{attribute 'linkalways'} 
{attribute 'no_explicit_call' := 'This FB is a CLASS and must be accessed using methods or properties'}
{attribute 'enable_dynamic_creation'}
FUNCTION_BLOCK _ETcVnEstimationAlgorithm EXTENDS EnumDatatypeBase
VAR
	localData : ETcVnEstimationAlgorithm;
	activeData : REFERENCE TO ETcVnEstimationAlgorithm;
	enumBaseDatatype : _DINT(localData);
END_VAR

METHOD PRIVATE AddLocalEnumeration
VAR_INPUT
	Enumeration : T_MAXSTRING;
	Value : ETcVnEstimationAlgorithm;
END_VAR
AddEnumeration(Enumeration, Value);
END_METHOD

PROPERTY PUBLIC Address : PVOID
GET
Address := ADR(activeData);
END_GET
END_PROPERTY

METHOD PUBLIC ClearReference
VAR_INPUT
END_VAR
activeData REF= localData;
SetBaseDatatypeReference();
END_METHOD

METHOD PUBLIC Clone : I_Datatype
VAR
    pClone : POINTER TO _ETcVnEstimationAlgorithm;
END_VAR
pClone := __NEW(_ETcVnEstimationAlgorithm(InitialValue := Value));
Clone := pClone^;
END_METHOD

METHOD FB_init : BOOL
VAR_INPUT
	bInitRetains : BOOL; // if TRUE, the retain variables are initialized (warm start / cold start)
	bInCopyCode : BOOL;  // if TRUE, the instance afterwards gets moved into the copy code (online change)
	InitialValue : ETcVnEstimationAlgorithm;
END_VAR
localData := InitialValue;
AddBaseDatatype(enumBaseDatatype);
ClearReference();

AddLocalEnumeration('TCVN_EA_DEFAULT', ETcVnEstimationAlgorithm.TCVN_EA_DEFAULT);
AddLocalEnumeration('TCVN_EA_LMEDS', ETcVnEstimationAlgorithm.TCVN_EA_LMEDS);
AddLocalEnumeration('TCVN_EA_RANSAC', ETcVnEstimationAlgorithm.TCVN_EA_RANSAC);
AddLocalEnumeration('TCVN_EA_RHO', ETcVnEstimationAlgorithm.TCVN_EA_RHO);
END_METHOD

PROPERTY PUBLIC Identifier : T_MAXSTRING
GET
Identifier := 'ETcVnEstimationAlgorithm';
END_GET
END_PROPERTY

METHOD IsEnumeratorValueEqual : BOOL
VAR_INPUT
	Enumerator : I_KeyValueForwardEnumerator;
END_VAR
VAR
	storedValue : ETcVnEstimationAlgorithm;
END_VAR
IF NOT Enumerator.TryGet(storedValue) THEN
	RETURN;
END_IF

IsEnumeratorValueEqual := storedValue = activeData;
END_METHOD

METHOD PUBLIC MakeReferenceTo
VAR_INPUT
	ReferenceTarget : REFERENCE TO ETcVnEstimationAlgorithm;
END_VAR
activeData REF= ReferenceTarget;
SetBaseDatatypeReference();
END_METHOD

METHOD PROTECTED SetBaseDatatypeReference
VAR_INPUT
END_VAR
enumBaseDatatype.MakeReferenceTo(activeData);
END_METHOD

PROPERTY PUBLIC Size : UDINT
GET
Size := SIZEOF(activeData);
END_GET
END_PROPERTY

METHOD TryMakeReferenceTo : BOOL
VAR_INPUT
	Target : I_Datatype;
END_VAR
VAR
	targetAsEnum : I_EnumDatatype;
	pTargetData : POINTER TO ETcVnEstimationAlgorithm;
END_VAR
IF NOT Target.TryResolveAsEnumDatatype(targetAsEnum) THEN
	RETURN;
END_IF

IF targetAsEnum.Identifier <> Identifier THEN
	RETURN;
END_IF

pTargetData := Target.Address;
activeData REF= pTargetData^;
SetBaseDatatypeReference();
TryMakeReferenceTo := TRUE;
END_METHOD

PROPERTY PUBLIC Value : ETcVnEstimationAlgorithm
GET
Value := activeData;
END_GET
SET
activeData := Value;
END_SET
END_PROPERTY

END_FUNCTION_BLOCK

(* stored: Version 1.1.0.1, ProductVersion 3.1.4024.12
   POU _ETcVnEstimationAlgorithm: Id {e59bbdbe-7dfb-472a-899c-8f3a9645b6cd}, SpecialFunc None
   Folder Constructor: Id {69b6ce92-ee4b-4402-890e-e10167038869}
   Folder Private: Id {ac9322c8-696d-4102-ad80-040769ac0943}
   Folder Protected: Id {330da5af-c186-42ad-9bba-a84b052d31a7}
   Method AddLocalEnumeration: Id {844b4a35-3c88-44f5-871f-608cc5491dd9}
   Property Address: Id {8e77053f-eaa2-4120-877d-dd8f6885d39b}
   Get Get: Id {ee349de9-0a7c-4e65-9072-030aef8acab3}
   Method ClearReference: Id {ab6508d3-6fab-4a42-91a0-2ad6898304da}
   Method Clone: Id {58ac51bf-e618-42e8-98f0-93c0a3b9103d}
   Method FB_init: Id {9b7b25c3-1055-4ada-a60f-1200bd513c1e}
   Property Identifier: Id {5d197be4-cb02-4cde-9dea-3c8b976bff27}
   Get Get: Id {4c2e4fbc-c286-432d-8ceb-81d8de064ba3}
   Method IsEnumeratorValueEqual: Id {e14c1e2b-ec99-4969-a0b6-1eb3371da816}
   Method MakeReferenceTo: Id {350046f9-1fd8-4013-95ab-42bccfb0fbba}
   Method SetBaseDatatypeReference: Id {718bd049-cbe2-4d8a-9e6a-50367102116f}
   Property Size: Id {bb93c9e7-861a-49ea-a108-ad8d3e9d6176}
   Get Get: Id {a80cd4ae-3814-4ce1-83b0-78ed2100f148}
   Method TryMakeReferenceTo: Id {91a860ca-2207-4d76-8f0a-6a8169a5202b}
   Property Value: Id {c3a1dd3a-2dc2-4145-8a85-79c7e3dead9d}
   Get Get: Id {afa5e0c0-f3b9-42c3-9999-b232a0ac4d37}
   Set Set: Id {0a016413-4567-4e05-9516-cb387b4ddf38} *)
